{attribute 'linkalways'} 
{attribute 'no_explicit_call' := 'This FB is a CLASS and must be accessed using methods or properties'}
{attribute 'enable_dynamic_creation'}
FUNCTION_BLOCK KeyValueCollectionDisposedEvent EXTENDS KeyValueCollectionEvent IMPLEMENTS I_KeyValueCollectionDisposedEvent

END_FUNCTION_BLOCK

(* stored: Version 1.1.0.1, ProductVersion 3.1.4024.12
   POU KeyValueCollectionDisposedEvent: Id {546f5b05-7015-4eec-a284-ada20174395f}, SpecialFunc None *)
